// TIA Portal V16 export
// export: Created 2026-06-17T16:42:20.4382695Z, ExportSetting WithDefaults, DisplayName Totally Integrated Automation Portal, DisplayVersion V16 Update 8, DisplayName TIA Portal Version Control Interface, DisplayVersion V16 Update 8, DisplayName TIA Portal Openness, DisplayVersion V16 Update 8, DisplayName SINAMICS Startdrive Advanced, DisplayVersion V16, DisplayName SINAMICS Startdrive G130, G150, S120, S150, SINAMICS MV, S210, DisplayVersion V16, DisplayName SINAMICS Startdrive G110M, G120, G120C, G120D, G120P, DisplayVersion V16, DisplayName STEP 7 Professional, DisplayVersion V16 Update 8, DisplayName STEP 7 Safety, DisplayVersion V16 Update 7, DisplayName WinCC Advanced, DisplayVersion V16 Update 8
Screen "Operator_Login"  1280x800, Number=1
